// TIA Portal V18 program export: 0 tag tables, 0 data types, 0 data blocks, 1 code blocks (in call order from the OBs), 0 instance data blocks

ORGANIZATION_BLOCK "Main"   // OB1, LAD, ProgramCycle
TITLE = "Main Program Sweep (Cycle)"
{ S7_Optimized_Access := 'TRUE' }
VERSION : 0.1
// stored: AutoNumber true, IsIECCheckEnabled false, SetENOAutomatically false
   VAR_INPUT
      Initial_Call : Bool;   // Initial call of this OB
      Remanence : Bool;   // =True, if remanent data are available
   END_VAR
BEGIN

REGION Network 1: Network2_comment
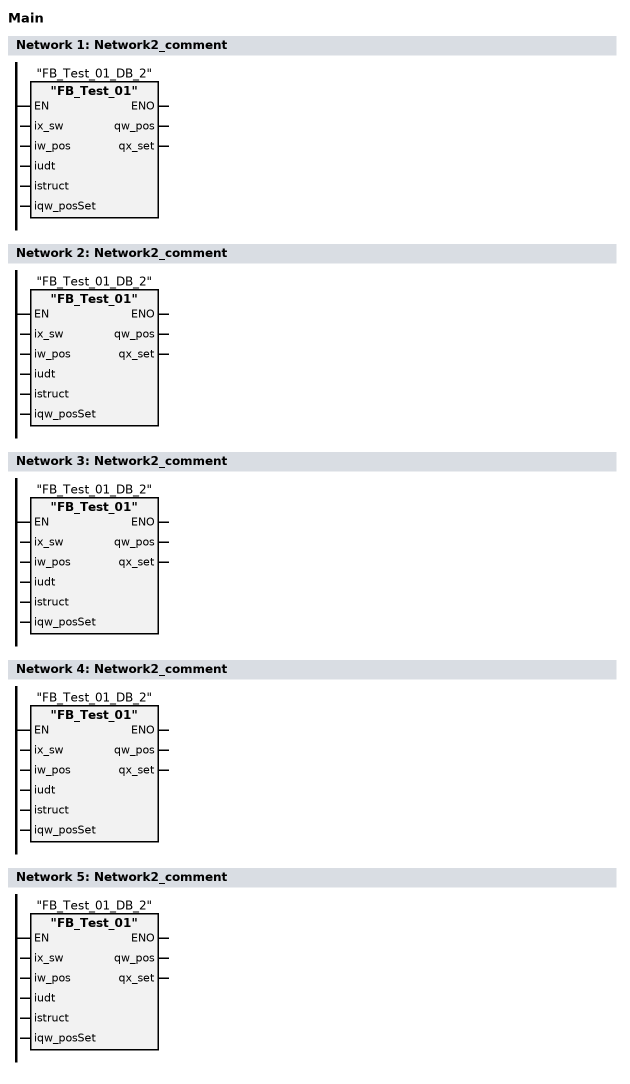
   RUNG wire#powerrail
      "FB_Test_01_DB_2"(ix_sw :=, iw_pos :=, iudt :=, istruct :=, iqw_posSet :=, qw_pos =>, qx_set =>)
   END_RUNG
   // the same network as SCL:
   "FB_Test_01_DB_2"();   // "FB_Test_01"
END_REGION

REGION Network 2: Network2_comment
   RUNG wire#powerrail
      "FB_Test_01_DB_2"(ix_sw :=, iw_pos :=, iudt :=, istruct :=, iqw_posSet :=, qw_pos =>, qx_set =>)
   END_RUNG
   // the same network as SCL:
   "FB_Test_01_DB_2"();   // "FB_Test_01"
END_REGION

REGION Network 3: Network2_comment
   RUNG wire#powerrail
      "FB_Test_01_DB_2"(ix_sw :=, iw_pos :=, iudt :=, istruct :=, iqw_posSet :=, qw_pos =>, qx_set =>)
   END_RUNG
   // the same network as SCL:
   "FB_Test_01_DB_2"();   // "FB_Test_01"
END_REGION

REGION Network 4: Network2_comment
   RUNG wire#powerrail
      "FB_Test_01_DB_2"(ix_sw :=, iw_pos :=, iudt :=, istruct :=, iqw_posSet :=, qw_pos =>, qx_set =>)
   END_RUNG
   // the same network as SCL:
   "FB_Test_01_DB_2"();   // "FB_Test_01"
END_REGION

REGION Network 5: Network2_comment
   RUNG wire#powerrail
      "FB_Test_01_DB_2"(ix_sw :=, iw_pos :=, iudt :=, istruct :=, iqw_posSet :=, qw_pos =>, qx_set =>)
   END_RUNG
   // the same network as SCL:
   "FB_Test_01_DB_2"();   // "FB_Test_01"
END_REGION
END_ORGANIZATION_BLOCK
